TYPE RTU_THT :
STRUCT
	Temp : REAL;
	RH : REAL;
	Temp_OOR : BOOL;
	RH_OOR : BOOL;
	CommsError : BOOL;
	CommsErrorCode : INT;
END_STRUCT
END_TYPE

(* stored: Version 1.1.0.1, ProductVersion 3.1.4024.12
   DUT RTU_THT: Id {f1103569-bfc1-4133-8d75-249cdf83790a} *)
